// TwinCAT 3 PLC project PLC_Interpolation_Library
// Title: PLC_Interpolation_Library
// Company: Chua Siang Poh
// Author: Chua Siang Poh
// ProjectVersion: 1.0
// Description: A simple library to enable you to use the NCI package to do PLC interpolation.
// ProgramVersion: 3.1.4020.10
// libraries:
//   Tc2_MC2, * (Beckhoff Automation GmbH)
//   Tc2_PlcInterpolation, * (Beckhoff Automation GmbH)
//   Tc2_Standard, * (Beckhoff Automation GmbH)
//   Tc2_System, * (Beckhoff Automation GmbH)
//   Tc3_Interfaces, * (Beckhoff Automation GmbH)
//   Tc3_Module, * (Beckhoff Automation GmbH)
// project tree:
//   Custom Datatypes/ Interpolation_FunctionResult.TcDUT, POSITION.TcDUT
//   / INTERPOLATION_CHANNEL.TcPOU, PLC_Interpolation_Parameters.TcGVL
//   Version/ Global_Version.TcGVL
// (motion and I/O tree: see PLC project motion_library)
// real-time tasks:
//   TASK PlcTask: cycle T#10ms, priority 20, ADS port 350

// ---- Custom Datatypes/Interpolation_FunctionResult.TcDUT
TYPE Interpolation_FunctionResult :
(
	Interpolation_OK := -1,
	Interpolation_Busy := 0,
	Interpolation_Error,
	Interpolation_OutOfBounds,
	Interpolation_Assignment_Cannot_Be_Same,
	Interpolation_Aborted
);
END_TYPE

// ---- Custom Datatypes/POSITION.TcDUT
TYPE POSITION :
STRUCT
	X : LREAL;
	Y : LREAL;
	Z : LREAL;
END_STRUCT
END_TYPE

// ---- PLC_Interpolation_Parameters.TcGVL
VAR_GLOBAL CONSTANT
	MAX_DIMENSIONS : INT := 3; (*Valid values are 1, 2, 3*)
END_VAR

// ---- Version/Global_Version.TcGVL
// This function has been automatically generated from the project information.
VAR_GLOBAL CONSTANT
	{attribute 'const_non_replaced'}
	stLibVersion_PLC_Interpolation_Library : ST_LibVersion := (iMajor := 1, iMinor := 0, iBuild := 0, iRevision := 0, sVersion := '1.0');
END_VAR

// ---- INTERPOLATION_CHANNEL.TcPOU
FUNCTION_BLOCK FINAL INTERPOLATION_CHANNEL
VAR_INPUT
END_VAR
VAR_OUTPUT
END_VAR
VAR
	MAIN_AXIS 	: ARRAY [1..MAX_DIMENSIONS] OF AXIS_REF;
	fbPower 	: ARRAY [1..MAX_DIMENSIONS] OF MC_POWER;
	fbReset 	: ARRAY [1..MAX_DIMENSIONS] OF MC_RESET;
	fbHome		: ARRAY	[1..MAX_DIMENSIONS] OF MC_HOME;
	fbMoveA 	: ARRAY [1..MAX_DIMENSIONS] OF MC_MOVEABSOLUTE;
	fbMoveR 	: ARRAY [1..MAX_DIMENSIONS] OF MC_MOVERELATIVE;
	fbJog		: ARRAY [1..MAX_DIMENSIONS] OF MC_JOG;
	fbHalt	 	: ARRAY [1..MAX_DIMENSIONS] OF MC_HALT;
	i			: INT;
END_VAR

;

METHOD PUBLIC On : Interpolation_FunctionResult
VAR_INPUT
	AXIS 		: INT;
	ENABLE_FW	: BOOL;
	ENABLE_BW	: BOOL;
	OVERRIDE 	: LREAL;
END_VAR
IF AXIS > MAX_DIMENSIONS OR AXIS < 1 THEN 
	On := Interpolation_FunctionResult.Interpolation_OutOfBounds;
ELSE
	fbPower[AXIS](
		Axis:= AXIS[AXIS].AXIS, 
		Enable:= TRUE, 
		Enable_Positive:= ENABLE_FW, 
		Enable_Negative:= ENABLE_BW, 
		Override:= OVERRIDE );
	IF fbPower[AXIS].Error THEN
		On := Interpolation_FunctionResult.Interpolation_Error;
	ELSIF fbPower[AXIS].Status THEN
		On := Interpolation_FunctionResult.Interpolation_OK;
	ELSE
		On := Interpolation_FunctionResult.Interpolation_Busy;
	END_IF
END_IF
END_METHOD

METHOD PUBLIC On_All : Interpolation_FunctionResult
VAR_INPUT
END_VAR
VAR
	n : INT;
	m : INT;
END_VAR
m := 0;
FOR n := 1 TO MAX_DIMENSIONS BY 1 DO
		fbPower[n](
		Axis:= MAIN_AXIS[n], 
		Enable:= TRUE, 
		Enable_Positive:= TRUE, 
		Enable_Negative:= TRUE, 
		Override:= 100 );
	IF fbPower[n].Error THEN
		On_All := Interpolation_FunctionResult.Interpolation_Error;
	ELSIF fbPower[n].Status THEN
		m := m + 1;
	END_IF
END_FOR
IF m >= MAX_DIMENSIONS THEN
	On_All := Interpolation_FunctionResult.Interpolation_OK;;
ELSE
	On_All := Interpolation_FunctionResult.Interpolation_Busy;
END_IF
END_METHOD

METHOD PUBLIC ASSIGN : Interpolation_FunctionResult
VAR_INPUT
	X : INT;
	Y : INT;
	Z : INT;
END_VAR
IF X < 1 OR X > MAX_DIMENSIONS THEN
	ASSIGN := Interpolation_FunctionResult.Interpolation_OutOfBounds;
END_IF
IF Y < 1 OR Y > MAX_DIMENSIONS THEN
	ASSIGN := Interpolation_FunctionResult.Interpolation_OutOfBounds;
END_IF
IF Z < 1 OR Z > MAX_DIMENSIONS THEN
	ASSIGN := Interpolation_FunctionResult.Interpolation_OutOfBounds;
END_IF
IF X = Y OR Y = Z OR Z = X THEN
	ASSIGN := Interpolation_FunctionResult.Interpolation_Assignment_Cannot_Be_Same;
END_IF
END_METHOD

END_FUNCTION_BLOCK
